{attribute 'qualified_only'}
{attribute 'strict'}
{attribute 'to_string'}
TYPE E_CilinderZuignapStatus :
(
	enum_member := 0
);
END_TYPE

(* stored: Version 1.1.0.1
   DUT E_CilinderZuignapStatus: Id {098901e3-5b1d-4fe9-9362-d2f1e0b6e1f1} *)
